FUNCTION_BLOCK FBSelection IMPLEMENTS ISelection
VAR_INPUT
END_VAR
VAR_OUTPUT
END_VAR
VAR
END_VAR

{warning 'add method implementation '}
METHOD TargetConverter : INT
VAR_INPUT
	sTargetName : STRING;	
END_VAR
VAR_OUTPUT
	TargetConverter_output : INT;	
END_VAR

VAR
	nTemp: INT;
	nVar: INT;
	bVar1: BOOL;
	bVar3: BOOL;
	bVar2: BOOL;
END_VAR
IF sTargetName = 'R1' THEN
	nTemp := 0;
ELSIF sTargetName = 'R2' THEN
	nTemp := 1;
ELSIF sTargetName = 'R3' THEN
	nTemp := 2;
ELSIF sTargetName = 'R4' THEN
	nTemp := 3;
ELSIF sTargetName = 'R5' THEN
	nTemp := 4;
ELSIF sTargetName = 'AA1' THEN
	nTemp := 5;
ELSIF sTargetName = 'AA2' THEN
	nTemp := 6;
ELSIF sTargetName = 'DCM' THEN
	nTemp := 7;
ELSIF sTargetName = 'MVB' THEN
	nTemp := 8;
ELSIF sTargetName = 'RV_50L' THEN
	nTemp := 10;
ELSIF sTargetName = 'MVA 25L' or sTargetName = 'MVA' THEN
	nTemp := 9;
ELSIF sTargetName = 'RV_25L' THEN
	nTemp := 11;
ELSIF sTargetName = 'Fill In' THEN
	nTemp := 12;
ELSIF sTargetName = 'Flash' THEN
	nTemp := 13;
ELSE
	nTemp := 14;	
END_IF

TargetConverter_output := nTemp;
END_METHOD

END_FUNCTION_BLOCK

(* stored: Version 1.1.0.1, ProductVersion 3.1.4024.5
   POU FBSelection: Id {d3e65dcb-c79d-4220-964a-13ed148d42f5}, SpecialFunc None
   Method TargetConverter: Id {86fa9da8-8495-4eaf-a2e9-48f9bffb3873} *)
